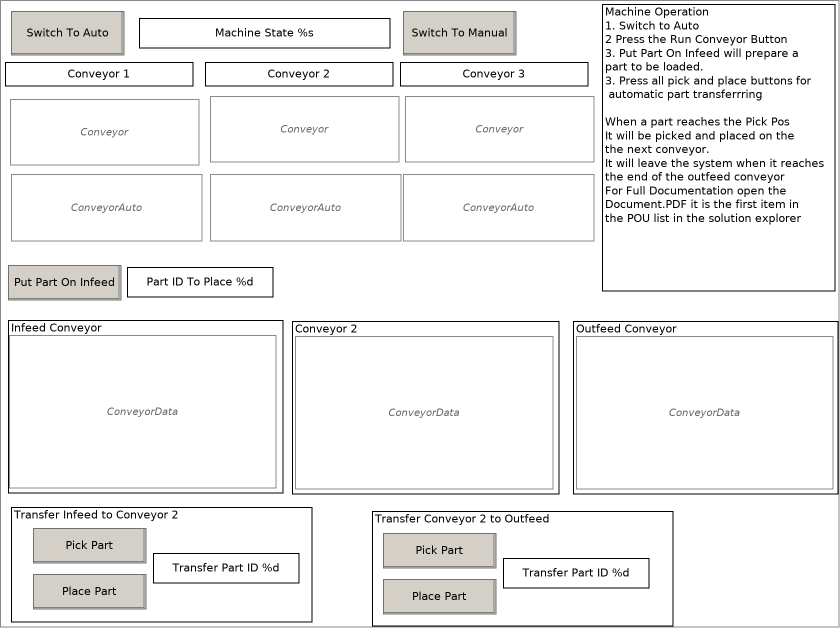
VISUALIZATION V_OOP_Conveyor  // 840x628
    Group (11,507 301x115)
        Rectangle (0,0 301x115), "Transfer Infeed to Conveyor 2"
        Button (22,21 113x35), "Pick Part", pressed state: MAIN.fbOOPConveyor.bPickPart
            toggle MAIN.fbOOPConveyor.bPickPart
        Rectangle (142,46 146x30), "Transfer Part ID %d", text variable: MAIN.fbOOPConveyor.fbTransfer1.stPart.iIDNumber
        Button (22,67 113x35), "Place Part", pressed state: MAIN.fbOOPConveyor.bPlacePart
            toggle MAIN.fbOOPConveyor.bPlacePart
    Button (11,11 113x44), "Switch To Auto"
        OnMouseDown: execute { MAIN.fbOOPConveyor.eMachineState := E_SwitchingToAuto; }
    Button (403,11 113x44), "Switch To Manual"
        OnMouseDown: execute { MAIN.fbOOPConveyor.eMachineState := E_SwitchingToManual; }
    Rectangle (139,18 251x30), "Machine State %s", text variable: MAIN.fbOOPConveyor.eMachineState
    Frame (10,99 189x66)
        shows Conveyor(bJogFwd := MAIN.fbOOPConveyor.bJogFwd, bJogBwd := MAIN.fbOOPConveyor.bJogBwd, fSpeed := MAIN.fbOOPConveyor.AxisRef[1].NcToPlc.ActVelo)
    Rectangle (5,62 188x24), "Conveyor 1"
    Frame (210,96 189x66)
        shows Conveyor(bJogFwd := MAIN.fbOOPConveyor.bJogFwd, bJogBwd := MAIN.fbOOPConveyor.bJogBwd, fSpeed := MAIN.fbOOPConveyor.iAnalogValue)
    Rectangle (205,62 188x24), "Conveyor 2"
    Frame (405,96 189x66)
        shows Conveyor(bJogFwd := MAIN.fbOOPConveyor.bJogFwd, bJogBwd := MAIN.fbOOPConveyor.bJogBwd, fSpeed := MAIN.fbOOPConveyor.AxisRef[2].NcToPlc.ActVelo)
    Rectangle (400,62 188x24), "Conveyor 3"
    Frame (11,174 191x67)
        shows ConveyorAuto(bRunConveyor := MAIN.fbOOPConveyor.bRunConveyor, fActualSpeed := MAIN.fbOOPConveyor.AxisRef[1].NcToPlc.ActVelo, fCmdSpeed := MAIN.fbOOPConveyor.fConveyorCmdSpeed)
    Button (8,265 113x35), "Put Part On Infeed", pressed state: MAIN.fbOOPConveyor.bPartPresent
        toggle MAIN.fbOOPConveyor.bPartPresent
    Frame (210,174 191x67)
        shows ConveyorAuto(bRunConveyor := MAIN.fbOOPConveyor.bRunConveyor, fActualSpeed := MAIN.fbOOPConveyor.fbConveyor2.fCurrentSpeed, fCmdSpeed := MAIN.fbOOPConveyor.fConveyorCmdSpeed)
    Rectangle (127,267 146x30), "Part ID To Place %d", text variable: arrParts[1].iIDNumber
    Group (292,321 267x173)
        Rectangle (0,0 267x173), "Conveyor 2"
        Frame (3,15 258x153)
            shows ConveyorData(fbConveyor := MAIN.fbOOPConveyor.fbConveyor2)
    Frame (403,174 191x67)
        shows ConveyorAuto(bRunConveyor := MAIN.fbOOPConveyor.bRunConveyor, fActualSpeed := MAIN.fbOOPConveyor.fbConveyor3.fCurrentSpeed, fCmdSpeed := MAIN.fbOOPConveyor.fConveyorCmdSpeed)
    Rectangle (8,320 275x173), "Infeed Conveyor"
    Frame (9,335 267x153)
        shows ConveyorData(fbConveyor := MAIN.fbOOPConveyor.fbInfeedConveyor)
    Group (372,511 301x115)
        Rectangle (0,0 301x115), "Transfer Conveyor 2 to Outfeed"
        Button (11,22 113x35), "Pick Part", pressed state: MAIN.fbOOPConveyor.bPickPart2
            toggle MAIN.fbOOPConveyor.bPickPart2
        Rectangle (131,47 146x30), "Transfer Part ID %d", text variable: MAIN.fbOOPConveyor.fbTransfer2.stPart.iIDNumber
        Button (11,68 113x35), "Place Part", pressed state: MAIN.fbOOPConveyor.bPlacePart2
            toggle MAIN.fbOOPConveyor.bPlacePart2
    Group (573,321 265x173)
        Rectangle (0,0 265x173), "Outfeed Conveyor"
        Frame (3,15 257x153)
            shows ConveyorData(fbConveyor := MAIN.fbOOPConveyor.fbConveyor3)
    Rectangle (602,4 233x287), "Machine Operation 1. Switch to Auto 2 Press the Run Conveyor Button 3. Put Part On Infeed will prepare a part to be loaded. 3. Press all pick and place buttons for automatic part transferrring When a part reaches the Pick Pos It will be picked and placed on the the next conveyor. It will leave the system when it reaches the end of the outfeed conveyor For Full Documentation open the Document.PDF it is the first item in the POU list in the solution explorer"
END_VISUALIZATION

(* stored: Version 1.1.0.1, ProductVersion 3.1.4024.11
   Visu V_OOP_Conveyor: Id {0377b294-8919-45f3-868f-aad55e68f189} *)
